// ---- DUTs/IO/Boxes/EQ2339_4CF33DED.TcDUT
{attribute 'GeneratedUsingTerminal: EQ2339-0022-0016'}
{attribute addProperty BoxType "EQ2339-0022-0016"}
{attribute addProperty Description "EQ2339-0022 16 Ch. Dig. Input/Output 24V, 0,5A, M12"}
{attribute addProperty Physics "YY"}
{attribute addProperty Id "Channel_1AT %I*Channel_830843C11Channel_2AT %I*Channel_830843C11Channel_3AT %I*Channel_830843C11Channel_4AT %I*Channel_830843C11Channel_5AT %I*Channel_830843C11Channel_6AT %I*Channel_830843C11Channel_7AT %I*Channel_830843C11Channel_8AT %I*Channel_830843C11Channel_9AT %I*Channel_830843C11Channel_10AT %I*Channel_830843C11Channel_11AT %I*Channel_830843C11Channel_12AT %I*Channel_830843C11Channel_13AT %I*Channel_830843C11Channel_14AT %I*Channel_830843C11Channel_15AT %I*Channel_830843C11Channel_16AT %I*Channel_830843C11Channel_17AT %Q*Channel_42CA91F71Channel_18AT %Q*Channel_42CA91F71Channel_19AT %Q*Channel_42CA91F71Channel_20AT %Q*Channel_42CA91F71Channel_21AT %Q*Channel_42CA91F71Channel_22AT %Q*Channel_42CA91F71Channel_23AT %Q*Channel_42CA91F71Channel_24AT %Q*Channel_42CA91F71Channel_25AT %Q*Channel_42CA91F71Channel_26AT %Q*Channel_42CA91F71Channel_27AT %Q*Channel_42CA91F71Channel_28AT %Q*Channel_42CA91F71Channel_29AT %Q*Channel_42CA91F71Channel_30AT %Q*Channel_42CA91F71Channel_31AT %Q*Channel_42CA91F71Channel_32AT %Q*Channel_42CA91F71WcStateAT %I*WcState_9091E0EB2InfoDataAT %I*InfoData_6F19DB2B2"}
{attribute addProperty CRC "1291009517"}
{attribute addProperty Size "36"}
TYPE EQ2339_4CF33DED EXTENDS EtcSlaveBoxBase_77A0E4A7 :
STRUCT
	{attribute addProperty Name "Channel_1"}
	Channel_1 : Channel_830843C1;
	{attribute addProperty Name "Channel_2"}
	Channel_2 : Channel_830843C1;
	{attribute addProperty Name "Channel_3"}
	Channel_3 : Channel_830843C1;
	{attribute addProperty Name "Channel_4"}
	Channel_4 : Channel_830843C1;
	{attribute addProperty Name "Channel_5"}
	Channel_5 : Channel_830843C1;
	{attribute addProperty Name "Channel_6"}
	Channel_6 : Channel_830843C1;
	{attribute addProperty Name "Channel_7"}
	Channel_7 : Channel_830843C1;
	{attribute addProperty Name "Channel_8"}
	Channel_8 : Channel_830843C1;
	{attribute addProperty Name "Channel_9"}
	Channel_9 : Channel_830843C1;
	{attribute addProperty Name "Channel_10"}
	Channel_10 : Channel_830843C1;
	{attribute addProperty Name "Channel_11"}
	Channel_11 : Channel_830843C1;
	{attribute addProperty Name "Channel_12"}
	Channel_12 : Channel_830843C1;
	{attribute addProperty Name "Channel_13"}
	Channel_13 : Channel_830843C1;
	{attribute addProperty Name "Channel_14"}
	Channel_14 : Channel_830843C1;
	{attribute addProperty Name "Channel_15"}
	Channel_15 : Channel_830843C1;
	{attribute addProperty Name "Channel_16"}
	Channel_16 : Channel_830843C1;
	{attribute addProperty Name "Channel_17"}
	Channel_17 : Channel_42CA91F7;
	{attribute addProperty Name "Channel_18"}
	Channel_18 : Channel_42CA91F7;
	{attribute addProperty Name "Channel_19"}
	Channel_19 : Channel_42CA91F7;
	{attribute addProperty Name "Channel_20"}
	Channel_20 : Channel_42CA91F7;
	{attribute addProperty Name "Channel_21"}
	Channel_21 : Channel_42CA91F7;
	{attribute addProperty Name "Channel_22"}
	Channel_22 : Channel_42CA91F7;
	{attribute addProperty Name "Channel_23"}
	Channel_23 : Channel_42CA91F7;
	{attribute addProperty Name "Channel_24"}
	Channel_24 : Channel_42CA91F7;
	{attribute addProperty Name "Channel_25"}
	Channel_25 : Channel_42CA91F7;
	{attribute addProperty Name "Channel_26"}
	Channel_26 : Channel_42CA91F7;
	{attribute addProperty Name "Channel_27"}
	Channel_27 : Channel_42CA91F7;
	{attribute addProperty Name "Channel_28"}
	Channel_28 : Channel_42CA91F7;
	{attribute addProperty Name "Channel_29"}
	Channel_29 : Channel_42CA91F7;
	{attribute addProperty Name "Channel_30"}
	Channel_30 : Channel_42CA91F7;
	{attribute addProperty Name "Channel_31"}
	Channel_31 : Channel_42CA91F7;
	{attribute addProperty Name "Channel_32"}
	Channel_32 : Channel_42CA91F7;
	{attribute addProperty Name "WcState"}
	WcState : WcState_9091E0EB;
	{attribute addProperty Name "InfoData"}
	InfoData : InfoData_6F19DB2B;
END_STRUCT
END_TYPE

// ---- DUTs/IO/Boxes/EQ2809_2B6483BD.TcDUT
{attribute 'GeneratedUsingTerminal: EQ2809-0022-0016'}
{attribute addProperty BoxType "EQ2809-0022-0016"}
{attribute addProperty Description "EQ2809-0022 16 Ch. Dig. Output 24V, 0,5A, M12"}
{attribute addProperty Physics "YY"}
{attribute addProperty Id "Channel_1AT %Q*Channel_42CA91F71Channel_2AT %Q*Channel_42CA91F71Channel_3AT %Q*Channel_42CA91F71Channel_4AT %Q*Channel_42CA91F71Channel_5AT %Q*Channel_42CA91F71Channel_6AT %Q*Channel_42CA91F71Channel_7AT %Q*Channel_42CA91F71Channel_8AT %Q*Channel_42CA91F71Channel_9AT %Q*Channel_42CA91F71Channel_10AT %Q*Channel_42CA91F71Channel_11AT %Q*Channel_42CA91F71Channel_12AT %Q*Channel_42CA91F71Channel_13AT %Q*Channel_42CA91F71Channel_14AT %Q*Channel_42CA91F71Channel_15AT %Q*Channel_42CA91F71Channel_16AT %Q*Channel_42CA91F71WcStateAT %I*WcState_0B2B16F91InfoDataAT %I*InfoData_6F19DB2B2"}
{attribute addProperty CRC "728007613"}
{attribute addProperty Size "19"}
TYPE EQ2809_2B6483BD EXTENDS EtcSlaveBoxBase_77A0E4A7 :
STRUCT
	{attribute addProperty Name "Channel_1"}
	Channel_1 : Channel_42CA91F7;
	{attribute addProperty Name "Channel_2"}
	Channel_2 : Channel_42CA91F7;
	{attribute addProperty Name "Channel_3"}
	Channel_3 : Channel_42CA91F7;
	{attribute addProperty Name "Channel_4"}
	Channel_4 : Channel_42CA91F7;
	{attribute addProperty Name "Channel_5"}
	Channel_5 : Channel_42CA91F7;
	{attribute addProperty Name "Channel_6"}
	Channel_6 : Channel_42CA91F7;
	{attribute addProperty Name "Channel_7"}
	Channel_7 : Channel_42CA91F7;
	{attribute addProperty Name "Channel_8"}
	Channel_8 : Channel_42CA91F7;
	{attribute addProperty Name "Channel_9"}
	Channel_9 : Channel_42CA91F7;
	{attribute addProperty Name "Channel_10"}
	Channel_10 : Channel_42CA91F7;
	{attribute addProperty Name "Channel_11"}
	Channel_11 : Channel_42CA91F7;
	{attribute addProperty Name "Channel_12"}
	Channel_12 : Channel_42CA91F7;
	{attribute addProperty Name "Channel_13"}
	Channel_13 : Channel_42CA91F7;
	{attribute addProperty Name "Channel_14"}
	Channel_14 : Channel_42CA91F7;
	{attribute addProperty Name "Channel_15"}
	Channel_15 : Channel_42CA91F7;
	{attribute addProperty Name "Channel_16"}
	Channel_16 : Channel_42CA91F7;
	{attribute addProperty Name "WcState"}
	WcState : WcState_0B2B16F9;
	{attribute addProperty Name "InfoData"}
	InfoData : InfoData_6F19DB2B;
END_STRUCT
END_TYPE

// ---- DUTs/IO/Boxes/EQ3174_DCC78662.TcDUT
{attribute 'GeneratedUsingTerminal: EQ3174-0002-0016'}
{attribute addProperty BoxType "EQ3174-0002-0016"}
{attribute addProperty Description "EQ3174-0002 4Ch. Ana. Input +/-10V, 0-10V, 0/4-20mA configurable"}
{attribute addProperty Physics "YY"}
{attribute addProperty Id "AI_Standard_Channel_1AT %I*AI_Standard_Channel_A8DF64E310AI_Standard_Channel_2AT %I*AI_Standard_Channel_A8DF64E310AI_Standard_Channel_3AT %I*AI_Standard_Channel_A8DF64E310AI_Standard_Channel_4AT %I*AI_Standard_Channel_A8DF64E310WcStateAT %I*WcState_9091E0EB2InfoDataAT %I*InfoData_32EB74EA10"}
{attribute addProperty CRC "3704063586"}
{attribute addProperty Size "52"}
TYPE EQ3174_DCC78662 EXTENDS EtcSlaveBoxBase_77A0E4A7 :
STRUCT
	{attribute addProperty Name "AI_Standard_Channel_1"}
	AI_Standard_Channel_1 : AI_Standard_Channel_A8DF64E3;
	{attribute addProperty Name "AI_Standard_Channel_2"}
	AI_Standard_Channel_2 : AI_Standard_Channel_A8DF64E3;
	{attribute addProperty Name "AI_Standard_Channel_3"}
	AI_Standard_Channel_3 : AI_Standard_Channel_A8DF64E3;
	{attribute addProperty Name "AI_Standard_Channel_4"}
	AI_Standard_Channel_4 : AI_Standard_Channel_A8DF64E3;
	{attribute addProperty Name "WcState"}
	WcState : WcState_9091E0EB;
	{attribute addProperty Name "InfoData"}
	InfoData : InfoData_32EB74EA;
END_STRUCT
END_TYPE

// ---- DUTs/IO/Boxes/EQ3204_6CD7E119.TcDUT
{attribute 'GeneratedUsingTerminal: EQ3204-0002-0016'}
{attribute addProperty BoxType "EQ3204-0002-0016"}
{attribute addProperty Description "EQ3204-0002 4Ch. Ana. Input PT100 (RTD)"}
{attribute addProperty Physics "YY"}
{attribute addProperty Id "RTD_RTDInputs_Channel_1AT %I*RTD_RTDInputs_Channel_A8DF64E310RTD_RTDInputs_Channel_2AT %I*RTD_RTDInputs_Channel_A8DF64E310RTD_RTDInputs_Channel_3AT %I*RTD_RTDInputs_Channel_A8DF64E310RTD_RTDInputs_Channel_4AT %I*RTD_RTDInputs_Channel_A8DF64E310WcStateAT %I*WcState_9091E0EB2InfoDataAT %I*InfoData_32EB74EA10"}
{attribute addProperty CRC "1826087193"}
{attribute addProperty Size "52"}
TYPE EQ3204_6CD7E119 EXTENDS EtcSlaveBoxBase_77A0E4A7 :
STRUCT
	{attribute addProperty Name "RTD_RTDInputs_Channel_1"}
	RTD_RTDInputs_Channel_1 : RTD_RTDInputs_Channel_A8DF64E3;
	{attribute addProperty Name "RTD_RTDInputs_Channel_2"}
	RTD_RTDInputs_Channel_2 : RTD_RTDInputs_Channel_A8DF64E3;
	{attribute addProperty Name "RTD_RTDInputs_Channel_3"}
	RTD_RTDInputs_Channel_3 : RTD_RTDInputs_Channel_A8DF64E3;
	{attribute addProperty Name "RTD_RTDInputs_Channel_4"}
	RTD_RTDInputs_Channel_4 : RTD_RTDInputs_Channel_A8DF64E3;
	{attribute addProperty Name "WcState"}
	WcState : WcState_9091E0EB;
	{attribute addProperty Name "InfoData"}
	InfoData : InfoData_32EB74EA;
END_STRUCT
END_TYPE

// ---- DUTs/IO/Boxes/EQ3204_AB25C3AC.TcDUT
{attribute 'GeneratedUsingTerminal: EQ3204-0002-0021'}
{attribute addProperty BoxType "EQ3204-0002-0021"}
{attribute addProperty Description "EQ3204-0002 4Ch. Ana. Input PT100 (RTD)"}
{attribute addProperty Physics "YY"}
{attribute addProperty Id "RTD_RTDInputs_Channel_1AT %I*AI_Standard_Channel_4A3944819RTD_RTDInputs_Channel_2AT %I*AI_Standard_Channel_4A3944819RTD_RTDInputs_Channel_3AT %I*AI_Standard_Channel_4A3944819RTD_RTDInputs_Channel_4AT %I*AI_Standard_Channel_4A3944819WcStateAT %I*WcState_9091E0EB2InfoDataAT %I*InfoData_32EB74EA10"}
{attribute addProperty CRC "2871378860"}
{attribute addProperty Size "48"}
TYPE EQ3204_AB25C3AC EXTENDS EtcSlaveBoxBase_77A0E4A7 :
STRUCT
	{attribute addProperty Name "RTD_RTDInputs_Channel_1"}
	RTD_RTDInputs_Channel_1 : AI_Standard_Channel_4A394481;
	{attribute addProperty Name "RTD_RTDInputs_Channel_2"}
	RTD_RTDInputs_Channel_2 : AI_Standard_Channel_4A394481;
	{attribute addProperty Name "RTD_RTDInputs_Channel_3"}
	RTD_RTDInputs_Channel_3 : AI_Standard_Channel_4A394481;
	{attribute addProperty Name "RTD_RTDInputs_Channel_4"}
	RTD_RTDInputs_Channel_4 : AI_Standard_Channel_4A394481;
	{attribute addProperty Name "WcState"}
	WcState : WcState_9091E0EB;
	{attribute addProperty Name "InfoData"}
	InfoData : InfoData_32EB74EA;
END_STRUCT
END_TYPE

// ---- DUTs/IO/Boxes/EQ3314_1CEB931C.TcDUT
{attribute 'GeneratedUsingTerminal: EQ3314-0002-0016'}
{attribute addProperty BoxType "EQ3314-0002-0016"}
{attribute addProperty Description "EQ3314-0002 4Ch. Ana. Input Thermocouple (TC)"}
{attribute addProperty Physics "YY"}
{attribute addProperty Id "TC_TCInputs_Channel_1AT %I*TC_TCInputs_Channel_A8DF64E310TC_TCInputs_Channel_2AT %I*TC_TCInputs_Channel_A8DF64E310TC_TCInputs_Channel_3AT %I*TC_TCInputs_Channel_A8DF64E310TC_TCInputs_Channel_4AT %I*TC_TCInputs_Channel_A8DF64E310WcStateAT %I*WcState_9091E0EB2InfoDataAT %I*InfoData_32EB74EA10"}
{attribute addProperty CRC "485200668"}
{attribute addProperty Size "52"}
TYPE EQ3314_1CEB931C EXTENDS EtcSlaveBoxBase_77A0E4A7 :
STRUCT
	{attribute addProperty Name "TC_TCInputs_Channel_1"}
	TC_TCInputs_Channel_1 : TC_TCInputs_Channel_A8DF64E3;
	{attribute addProperty Name "TC_TCInputs_Channel_2"}
	TC_TCInputs_Channel_2 : TC_TCInputs_Channel_A8DF64E3;
	{attribute addProperty Name "TC_TCInputs_Channel_3"}
	TC_TCInputs_Channel_3 : TC_TCInputs_Channel_A8DF64E3;
	{attribute addProperty Name "TC_TCInputs_Channel_4"}
	TC_TCInputs_Channel_4 : TC_TCInputs_Channel_A8DF64E3;
	{attribute addProperty Name "WcState"}
	WcState : WcState_9091E0EB;
	{attribute addProperty Name "InfoData"}
	InfoData : InfoData_32EB74EA;
END_STRUCT
END_TYPE

// ---- DUTs/IO/Boxes/EQ3314_E65CDB1C.TcDUT
{attribute 'GeneratedUsingTerminal: EQ3314-0002-0022'}
{attribute addProperty BoxType "EQ3314-0002-0022"}
{attribute addProperty Description "EQ3314-0002 4Ch. Ana. Input Thermocouple (TC)"}
{attribute addProperty Physics "YY"}
{attribute addProperty Id "TC_Inputs_Channel_1AT %I*AI_Standard_Channel_4A3944819TC_Inputs_Channel_2AT %I*AI_Standard_Channel_4A3944819TC_Inputs_Channel_3AT %I*AI_Standard_Channel_4A3944819TC_Inputs_Channel_4AT %I*AI_Standard_Channel_4A3944819WcStateAT %I*WcState_9091E0EB2InfoDataAT %I*InfoData_32EB74EA10"}
{attribute addProperty CRC "3864845084"}
{attribute addProperty Size "48"}
TYPE EQ3314_E65CDB1C EXTENDS EtcSlaveBoxBase_77A0E4A7 :
STRUCT
	{attribute addProperty Name "TC_Inputs_Channel_1"}
	TC_Inputs_Channel_1 : AI_Standard_Channel_4A394481;
	{attribute addProperty Name "TC_Inputs_Channel_2"}
	TC_Inputs_Channel_2 : AI_Standard_Channel_4A394481;
	{attribute addProperty Name "TC_Inputs_Channel_3"}
	TC_Inputs_Channel_3 : AI_Standard_Channel_4A394481;
	{attribute addProperty Name "TC_Inputs_Channel_4"}
	TC_Inputs_Channel_4 : AI_Standard_Channel_4A394481;
	{attribute addProperty Name "WcState"}
	WcState : WcState_9091E0EB;
	{attribute addProperty Name "InfoData"}
	InfoData : InfoData_32EB74EA;
END_STRUCT
END_TYPE

// ---- DUTs/IO/Devices/SyncUnitTask_2D604ED5.TcDUT
{attribute 'GeneratedUsingTerminal: IODEVICETYPE_ETHERCATPROT'}
{attribute addProperty BoxType "IODEVICETYPE_ETHERCATPROT"}
{attribute addProperty Id "WcStateAT %I*WcState_0B2B16F91InfoDataAT %I*InfoData_2A97D6CF8"}
{attribute addProperty CRC "761286357"}
{attribute addProperty Size "9"}
TYPE SyncUnitTask_2D604ED5 :
STRUCT
	{attribute addProperty Name "WcState"}
	WcState : WcState_0B2B16F9;
	{attribute addProperty Name "InfoData"}
	InfoData : InfoData_2A97D6CF;
END_STRUCT
END_TYPE

// ---- DUTs/IO/Devices/SyncUnitTasks_6FEB8257.TcDUT
{attribute 'GeneratedUsingTerminal: '}
{attribute addProperty BoxType ""}
{attribute addProperty Id "unreferencedAT %I*SyncUnitTask_2D604ED59PlcTaskAT %I*SyncUnitTask_2D604ED59"}
{attribute addProperty CRC "1877705303"}
{attribute addProperty Size "18"}
TYPE SyncUnitTasks_6FEB8257 :
STRUCT
	{attribute addProperty Name "unreferenced"}
	unreferenced : SyncUnitTask_2D604ED5;
	{attribute addProperty Name "PlcTask"}
	PlcTask : SyncUnitTask_2D604ED5;
END_STRUCT
END_TYPE

// ---- DUTs/IO/Devices/SyncUnits_99E584AF.TcDUT
{attribute 'GeneratedUsingTerminal: '}
{attribute addProperty BoxType ""}
{attribute addProperty Id "_defaultAT %I*SyncUnitTasks_6FEB825718"}
{attribute addProperty CRC "2581955759"}
{attribute addProperty Size "18"}
TYPE SyncUnits_99E584AF :
STRUCT
	{attribute addProperty Name "_default"}
	_default : SyncUnitTasks_6FEB8257;
END_STRUCT
END_TYPE

// ---- DUTs/IO/Topology/Beckhoff_EQ1xxxEK1122_E78E0C94.TcDUT
{attribute 'GeneratedUsingTerminal: EK1122-0000-0018'}
{attribute addProperty BoxType "EK1122-0000-0018"}
{attribute addProperty Id "Beckhoff_EQ1xxxsub_EK1100EK1100_1FC0878B2A_0001_EQ1008_0002_0016EQ1008_78E8D3DD12A_0002_EQ1008_0002_0017EQ1008_78E8D3DD12A_0003_EQ1008_0002_0018EQ1008_78E8D3DD12A_0004_EQ1809_0022_0016EQ1809_32157CFD20A_0005_EQ1809_0022_0018EQ1809_32157CFD20"}
{attribute addProperty CRC "3884846228"}
{attribute addProperty Size "78"}
{attribute addProperty Name "Beckhoff EQ1xxxEK1122"}
TYPE Beckhoff_EQ1xxxEK1122_E78E0C94 EXTENDS EK1122_1FC0878B :
STRUCT
	{attribute addProperty Name "Beckhoff EQ1xxxsub EK1100"}
	{attribute addProperty PreviousPort "Beckhoff EQ1xxxEK1122 : D"}
	Beckhoff_EQ1xxxsub_EK1100 : EK1100_1FC0878B;
	{attribute addProperty Name "A_0001(EQ1008-0002-0016)"}
	{attribute addProperty PreviousPort "Beckhoff EQ1xxxsub EK1100 : C"}
	A_0001_EQ1008_0002_0016 : EQ1008_78E8D3DD;
	{attribute addProperty Name "A_0002(EQ1008-0002-0017)"}
	{attribute addProperty PreviousPort "A_0001(EQ1008-0002-0016) : B"}
	A_0002_EQ1008_0002_0017 : EQ1008_78E8D3DD;
	{attribute addProperty Name "A_0003(EQ1008-0002-0018)"}
	{attribute addProperty PreviousPort "A_0002(EQ1008-0002-0017) : B"}
	A_0003_EQ1008_0002_0018 : EQ1008_78E8D3DD;
	{attribute addProperty Name "A_0004(EQ1809-0022-0016)"}
	{attribute addProperty PreviousPort "A_0003(EQ1008-0002-0018) : B"}
	A_0004_EQ1809_0022_0016 : EQ1809_32157CFD;
	{attribute addProperty Name "A_0005(EQ1809-0022-0018)"}
	{attribute addProperty PreviousPort "A_0004(EQ1809-0022-0016) : B"}
	A_0005_EQ1809_0022_0018 : EQ1809_32157CFD;
END_STRUCT
END_TYPE

// ---- DUTs/IO/Topology/Beckhoff_EQ1xxx_F67C323D.TcDUT
{attribute 'GeneratedUsingTerminal: EK1100-0000-0018'}
{attribute addProperty BoxType "EK1100-0000-0018"}
{attribute addProperty Id "Beckhoff_EQ1xxxEK1122Beckhoff_EQ1xxxEK1122_E78E0C9478"}
{attribute addProperty CRC "4135334461"}
{attribute addProperty Size "78"}
{attribute addProperty Name "Beckhoff EQ1xxx"}
TYPE Beckhoff_EQ1xxx_F67C323D EXTENDS EK1100_1FC0878B :
STRUCT
	{attribute addProperty Name "Beckhoff EQ1xxxEK1122"}
	{attribute addProperty PreviousPort "Beckhoff EQ1xxx : B"}
	Beckhoff_EQ1xxxEK1122 : Beckhoff_EQ1xxxEK1122_E78E0C94;
END_STRUCT
END_TYPE

// ---- DUTs/IO/Topology/Beckhoff_EQ2xxxEK1122_214B8BB9.TcDUT
{attribute 'GeneratedUsingTerminal: EK1122-0000-0018'}
{attribute addProperty BoxType "EK1122-0000-0018"}
{attribute addProperty Id "Beckhoff_EQ2xxxsub_EK1100EK1100_1FC0878B2A_0001_EQ2008_0002_0016EQ2008_E2806B9511A_0002_EQ2008_0002_0017EQ2008_E2806B9511A_0003_EQ2008_0002_0018EQ2008_E2806B9511A_0004_EQ2008_0002_0019EQ2008_E2806B9511A_0005_EQ2339_0022_0016EQ2339_4CF33DED36A_0006_EQ2339_0022_0017EQ2339_4CF33DED36A_0007_EQ2339_0022_0018EQ2339_4CF33DED36A_0008_EQ2339_0022_0019EQ2339_4CF33DED36A_0009_EQ2809_0022_0016EQ2809_2B6483BD19A_0010_EQ2809_0022_0017EQ2809_2B6483BD19A_0011_EQ2809_0022_0018EQ2809_2B6483BD19"}
{attribute addProperty CRC "558599097"}
{attribute addProperty Size "247"}
{attribute addProperty Name "Beckhoff EQ2xxxEK1122"}
TYPE Beckhoff_EQ2xxxEK1122_214B8BB9 EXTENDS EK1122_1FC0878B :
STRUCT
	{attribute addProperty Name "Beckhoff EQ2xxxsub EK1100"}
	{attribute addProperty PreviousPort "Beckhoff EQ2xxxEK1122 : D"}
	Beckhoff_EQ2xxxsub_EK1100 : EK1100_1FC0878B;
	{attribute addProperty Name "A_0001(EQ2008-0002-0016)"}
	{attribute addProperty PreviousPort "Beckhoff EQ2xxxsub EK1100 : C"}
	A_0001_EQ2008_0002_0016 : EQ2008_E2806B95;
	{attribute addProperty Name "A_0002(EQ2008-0002-0017)"}
	{attribute addProperty PreviousPort "A_0001(EQ2008-0002-0016) : B"}
	A_0002_EQ2008_0002_0017 : EQ2008_E2806B95;
	{attribute addProperty Name "A_0003(EQ2008-0002-0018)"}
	{attribute addProperty PreviousPort "A_0002(EQ2008-0002-0017) : B"}
	A_0003_EQ2008_0002_0018 : EQ2008_E2806B95;
	{attribute addProperty Name "A_0004(EQ2008-0002-0019)"}
	{attribute addProperty PreviousPort "A_0003(EQ2008-0002-0018) : B"}
	A_0004_EQ2008_0002_0019 : EQ2008_E2806B95;
	{attribute addProperty Name "A_0005(EQ2339-0022-0016)"}
	{attribute addProperty PreviousPort "A_0004(EQ2008-0002-0019) : B"}
	A_0005_EQ2339_0022_0016 : EQ2339_4CF33DED;
	{attribute addProperty Name "A_0006(EQ2339-0022-0017)"}
	{attribute addProperty PreviousPort "A_0005(EQ2339-0022-0016) : B"}
	A_0006_EQ2339_0022_0017 : EQ2339_4CF33DED;
	{attribute addProperty Name "A_0007(EQ2339-0022-0018)"}
	{attribute addProperty PreviousPort "A_0006(EQ2339-0022-0017) : B"}
	A_0007_EQ2339_0022_0018 : EQ2339_4CF33DED;
	{attribute addProperty Name "A_0008(EQ2339-0022-0019)"}
	{attribute addProperty PreviousPort "A_0007(EQ2339-0022-0018) : B"}
	A_0008_EQ2339_0022_0019 : EQ2339_4CF33DED;
	{attribute addProperty Name "A_0009(EQ2809-0022-0016)"}
	{attribute addProperty PreviousPort "A_0008(EQ2339-0022-0019) : B"}
	A_0009_EQ2809_0022_0016 : EQ2809_2B6483BD;
	{attribute addProperty Name "A_0010(EQ2809-0022-0017)"}
	{attribute addProperty PreviousPort "A_0009(EQ2809-0022-0016) : B"}
	A_0010_EQ2809_0022_0017 : EQ2809_2B6483BD;
	{attribute addProperty Name "A_0011(EQ2809-0022-0018)"}
	{attribute addProperty PreviousPort "A_0010(EQ2809-0022-0017) : B"}
	A_0011_EQ2809_0022_0018 : EQ2809_2B6483BD;
END_STRUCT
END_TYPE

// ---- DUTs/IO/Topology/Beckhoff_EQ2xxx_A19B669C.TcDUT
{attribute 'GeneratedUsingTerminal: EK1100-0000-0018'}
{attribute addProperty BoxType "EK1100-0000-0018"}
{attribute addProperty Id "Beckhoff_EQ2xxxEK1122Beckhoff_EQ2xxxEK1122_214B8BB9247"}
{attribute addProperty CRC "2711316124"}
{attribute addProperty Size "247"}
{attribute addProperty Name "Beckhoff EQ2xxx"}
TYPE Beckhoff_EQ2xxx_A19B669C EXTENDS EK1100_1FC0878B :
STRUCT
	{attribute addProperty Name "Beckhoff EQ2xxxEK1122"}
	{attribute addProperty PreviousPort "Beckhoff EQ2xxx : B"}
	Beckhoff_EQ2xxxEK1122 : Beckhoff_EQ2xxxEK1122_214B8BB9;
END_STRUCT
END_TYPE

// ---- DUTs/IO/Topology/Beckhoff_EQ3xxxEK1122_A1C56A21.TcDUT
{attribute 'GeneratedUsingTerminal: EK1122-0000-0018'}
{attribute addProperty BoxType "EK1122-0000-0018"}
{attribute addProperty Id "Beckhoff_EQ3xxxsub_EK1100EK1100_1FC0878B2A_0001_EQ3174_0002_0016EQ3174_DCC7866252A_0002_EQ3174_0002_0017EQ3174_DCC7866252A_0003_EQ3174_0002_0021EQ3174_DCC7866252A_0004_EQ3174_0002_0022EQ3174_DCC7866252A_0005_EQ3174_0002_0023EQ3174_DCC7866252A_0006_EQ3204_0002_0016EQ3204_6CD7E11952A_0007_EQ3204_0002_0017EQ3204_6CD7E11952A_0008_EQ3204_0002_0020EQ3204_6CD7E11952A_0009_EQ3204_0002_0021EQ3204_AB25C3AC48A_0010_EQ3204_0002_0022EQ3204_AB25C3AC48A_0011_EQ3314_0002_0016EQ3314_1CEB931C52A_0012_EQ3314_0002_0017EQ3314_1CEB931C52A_0013_EQ3314_0002_0021EQ3314_1CEB931C52A_0014_EQ3314_0002_0022EQ3314_E65CDB1C48"}
{attribute addProperty CRC "2714069537"}
{attribute addProperty Size "718"}
{attribute addProperty Name "Beckhoff EQ3xxxEK1122"}
TYPE Beckhoff_EQ3xxxEK1122_A1C56A21 EXTENDS EK1122_1FC0878B :
STRUCT
	{attribute addProperty Name "Beckhoff EQ3xxxsub EK1100"}
	{attribute addProperty PreviousPort "Beckhoff EQ3xxxEK1122 : D"}
	Beckhoff_EQ3xxxsub_EK1100 : EK1100_1FC0878B;
	{attribute addProperty Name "A_0001(EQ3174-0002-0016)"}
	{attribute addProperty PreviousPort "Beckhoff EQ3xxxsub EK1100 : C"}
	A_0001_EQ3174_0002_0016 : EQ3174_DCC78662;
	{attribute addProperty Name "A_0002(EQ3174-0002-0017)"}
	{attribute addProperty PreviousPort "A_0001(EQ3174-0002-0016) : B"}
	A_0002_EQ3174_0002_0017 : EQ3174_DCC78662;
	{attribute addProperty Name "A_0003(EQ3174-0002-0021)"}
	{attribute addProperty PreviousPort "A_0002(EQ3174-0002-0017) : B"}
	A_0003_EQ3174_0002_0021 : EQ3174_DCC78662;
	{attribute addProperty Name "A_0004(EQ3174-0002-0022)"}
	{attribute addProperty PreviousPort "A_0003(EQ3174-0002-0021) : B"}
	A_0004_EQ3174_0002_0022 : EQ3174_DCC78662;
	{attribute addProperty Name "A_0005(EQ3174-0002-0023)"}
	{attribute addProperty PreviousPort "A_0004(EQ3174-0002-0022) : B"}
	A_0005_EQ3174_0002_0023 : EQ3174_DCC78662;
	{attribute addProperty Name "A_0006(EQ3204-0002-0016)"}
	{attribute addProperty PreviousPort "A_0005(EQ3174-0002-0023) : B"}
	A_0006_EQ3204_0002_0016 : EQ3204_6CD7E119;
	{attribute addProperty Name "A_0007(EQ3204-0002-0017)"}
	{attribute addProperty PreviousPort "A_0006(EQ3204-0002-0016) : B"}
	A_0007_EQ3204_0002_0017 : EQ3204_6CD7E119;
	{attribute addProperty Name "A_0008(EQ3204-0002-0020)"}
	{attribute addProperty PreviousPort "A_0007(EQ3204-0002-0017) : B"}
	A_0008_EQ3204_0002_0020 : EQ3204_6CD7E119;
	{attribute addProperty Name "A_0009(EQ3204-0002-0021)"}
	{attribute addProperty PreviousPort "A_0008(EQ3204-0002-0020) : B"}
	A_0009_EQ3204_0002_0021 : EQ3204_AB25C3AC;
	{attribute addProperty Name "A_0010(EQ3204-0002-0022)"}
	{attribute addProperty PreviousPort "A_0009(EQ3204-0002-0021) : B"}
	A_0010_EQ3204_0002_0022 : EQ3204_AB25C3AC;
	{attribute addProperty Name "A_0011(EQ3314-0002-0016)"}
	{attribute addProperty PreviousPort "A_0010(EQ3204-0002-0022) : B"}
	A_0011_EQ3314_0002_0016 : EQ3314_1CEB931C;
	{attribute addProperty Name "A_0012(EQ3314-0002-0017)"}
	{attribute addProperty PreviousPort "A_0011(EQ3314-0002-0016) : B"}
	A_0012_EQ3314_0002_0017 : EQ3314_1CEB931C;
	{attribute addProperty Name "A_0013(EQ3314-0002-0021)"}
	{attribute addProperty PreviousPort "A_0012(EQ3314-0002-0017) : B"}
	A_0013_EQ3314_0002_0021 : EQ3314_1CEB931C;
	{attribute addProperty Name "A_0014(EQ3314-0002-0022)"}
	{attribute addProperty PreviousPort "A_0013(EQ3314-0002-0021) : B"}
	A_0014_EQ3314_0002_0022 : EQ3314_E65CDB1C;
END_STRUCT
END_TYPE

// ---- DUTs/IO/Topology/Beckhoff_EQ3xxx_A920B096.TcDUT
{attribute 'GeneratedUsingTerminal: EK1100-0000-0018'}
{attribute addProperty BoxType "EK1100-0000-0018"}
{attribute addProperty Id "Beckhoff_EQ3xxxEK1122Beckhoff_EQ3xxxEK1122_A1C56A21718"}
{attribute addProperty CRC "2837491862"}
{attribute addProperty Size "718"}
{attribute addProperty Name "Beckhoff EQ3xxx"}
TYPE Beckhoff_EQ3xxx_A920B096 EXTENDS EK1100_1FC0878B :
STRUCT
	{attribute addProperty Name "Beckhoff EQ3xxxEK1122"}
	{attribute addProperty PreviousPort "Beckhoff EQ3xxx : B"}
	Beckhoff_EQ3xxxEK1122 : Beckhoff_EQ3xxxEK1122_A1C56A21;
END_STRUCT
END_TYPE

// ---- DUTs/IO/Topology/EtherCAT_Master_EQxxxx_806C2CF0.TcDUT
{attribute 'GeneratedUsingTerminal: IODEVICETYPE_ETHERCATPROT'}
{attribute addProperty BoxType "IODEVICETYPE_ETHERCATPROT"}
{attribute addProperty Id "Beckhoff_EQ1xxxBeckhoff_EQ1xxx_F67C323D78Beckhoff_EQ2xxxBeckhoff_EQ2xxx_A19B669C247Beckhoff_EQ3xxxBeckhoff_EQ3xxx_A920B096718SyncUnitsSyncUnits_99E584AF18InputsInputs_25A0042B160OutputsOutputs_2397A10E106InfoDataInfoData_E68C61CD28"}
{attribute addProperty CRC "2154573040"}
{attribute addProperty Size "1355"}
{attribute addProperty Name "EtherCAT Master EQxxxx"}
TYPE EtherCAT_Master_EQxxxx_806C2CF0 EXTENDS EtcMasterBase_62654B43 :
STRUCT
	{attribute addProperty Name "Beckhoff EQ1xxx"}
	{attribute addProperty PreviousPort "EtherCAT Master EQxxxx : Master"}
	Beckhoff_EQ1xxx : Beckhoff_EQ1xxx_F67C323D;
	{attribute addProperty Name "Beckhoff EQ2xxx"}
	{attribute addProperty PreviousPort "Beckhoff EQ1xxx : C"}
	Beckhoff_EQ2xxx : Beckhoff_EQ2xxx_A19B669C;
	{attribute addProperty Name "Beckhoff EQ3xxx"}
	{attribute addProperty PreviousPort "Beckhoff EQ2xxx : C"}
	Beckhoff_EQ3xxx : Beckhoff_EQ3xxx_A920B096;
	{attribute addProperty Name "SyncUnits"}
	SyncUnits : SyncUnits_99E584AF;
	{attribute addProperty Name "Inputs"}
	Inputs : Inputs_25A0042B;
	{attribute addProperty Name "Outputs"}
	Outputs : Outputs_2397A10E;
	{attribute addProperty Name "InfoData"}
	InfoData : InfoData_E68C61CD;
END_STRUCT
END_TYPE

// ---- DUTs/IO/Base/EtcSlaveBase_82538BE2.TcDUT

TYPE EtcSlaveBase_82538BE2 :
STRUCT
END_STRUCT
END_TYPE

// ---- DUTs/IO/Base/EtcSlaveBase_82538BE2.TcDUT

TYPE EtcSlaveBase_82538BE2 :
STRUCT
END_STRUCT
END_TYPE

// ---- DUTs/IO/Base/EtcSlaveBase_82538BE2.TcDUT

TYPE EtcSlaveBase_82538BE2 :
STRUCT
END_STRUCT
END_TYPE

// ---- DUTs/IO/Base/EtcSlaveTerminalBase_947E5A46.TcDUT

{attribute clr[Container(Layout.Stack)]}
{attribute clr[Group(Layout.GroupBox)]}
{attribute addProperty PreviousPort "Unknown"}
TYPE EtcSlaveTerminalBase_947E5A46 EXTENDS EtcSlaveBase_82538BE2 :
STRUCT
END_STRUCT
END_TYPE

// ---- DUTs/IO/Base/EtcSlaveBoxBase_77A0E4A7.TcDUT

{attribute clr[Container(Layout.Stack)]}
{attribute clr[Group(Layout.GroupBox)]}
{attribute addProperty PreviousPort "Unknown"}
TYPE EtcSlaveBoxBase_77A0E4A7 EXTENDS EtcSlaveBase_82538BE2 :
STRUCT
END_STRUCT
END_TYPE

// ---- DUTs/IO/Base/EtcSlaveEndTerminalBase_866C7F0C.TcDUT

{attribute clr[Container(Layout.Stack)]}
{attribute clr[Group(Layout.GroupBox)]}
{attribute addProperty PreviousPort "Unknown"}
TYPE EtcSlaveEndTerminalBase_866C7F0C EXTENDS EtcSlaveBase_82538BE2 :
STRUCT
END_STRUCT
END_TYPE

// ---- DUTs/IO/Base/InputBase_8311D824.TcDUT

TYPE InputBase_8311D824 :
STRUCT
END_STRUCT
END_TYPE

// ---- DUTs/IO/Base/OutputBase_10CEE7DE.TcDUT

TYPE OutputBase_10CEE7DE :
STRUCT
END_STRUCT
END_TYPE

// ---- DUTs/IO/Base/EtcMasterBase_62654B43.TcDUT

TYPE EtcMasterBase_62654B43 :
STRUCT
END_STRUCT
END_TYPE

// ---- GVLs/GVL_iXlinker.TcGVL
{attribute 'qualified_only'}
VAR_GLOBAL
		EtherCAT_Master_EQxxxx : EtherCAT_Master_EQxxxx_806C2CF0;
END_VAR

// ---- POUs/MAIN.TcPOU
PROGRAM MAIN
VAR
END_VAR

END_PROGRAM
